{attribute addProperty BoxType "EL3692-0000-0017"}
{attribute addProperty Id "ValueAT %I*REAL324"}
{attribute addProperty CRC "1594033361"}
{attribute addProperty SizeInBites "32"}
{attribute addProperty SizeInBytes "4"}
TYPE SAI_Inputs_Real_Channel_5F0304D1 :
STRUCT
	{attribute addProperty Name "Value"}
	Value AT %I* : REAL;
END_STRUCT
END_TYPE

(* stored: Version 1.2.0.0, ProductVersion 3.1.4024.9
   DUT SAI_Inputs_Real_Channel_5F0304D1: Id {6d69279c-1b50-4a0d-9684-7e1f208186d5} *)
